// Copyright (c) 2024 Loupe (https://loupe.team), provided under the MIT License.

INTERFACE IPLCopenGroup

METHOD AbortPreviousCommands : BOOL
VAR_INPUT
    newCommand : IPLCopenCommand;
END_VAR
END_METHOD

END_INTERFACE

(* stored: Version 1.1.0.1
   Itf IPLCopenGroup: Id {b35eb493-5dd7-45b9-9e67-a673072a60b4}
   Method AbortPreviousCommands: Id {33d62d2b-227e-4998-b717-c18b2f1e35eb} *)
